// TIA Portal V17 export
// export: Created 2022-03-12T16:05:15.1481305Z, ExportSetting WithDefaults, DisplayName Totally Integrated Automation Portal, DisplayVersion V17, DisplayName TIA Portal Openness, DisplayVersion V17, DisplayName TIA Portal Version Control Interface, DisplayVersion V17, DisplayName STEP 7 Professional, DisplayVersion V17, DisplayName STEP 7 Safety, DisplayVersion V17, DisplayName WinCC Advanced / Unified PC, DisplayVersion V17
FUNCTION_BLOCK "UN_02_PackML"   // FB31622, LAD
TITLE = UN_02_PackML
{ S7_Optimized_Access := 'TRUE' }
AUTHOR : tech.team.motioncontrol@siemens.com
FAMILY : CPG
VERSION : 1.0
// Support: tech.team.motioncontrol@siemens.com
// Fax: +49 (0) 9131/98-1297
// stored: AutoNumber true, IsIECCheckEnabled false, IsRetainMemResEnabled false, MemoryReserve 100, SetENOAutomatically false, UDAEnableTagReadback false
   VAR
      statLanguageSelectedOld { ExternalAccessible := 'False'; ExternalVisible := 'False'; ExternalWritable := 'False'} : Int := -1;
      statPackML_CMD_SC { ExternalAccessible := 'False'; ExternalVisible := 'False'; ExternalWritable := 'False'} : Bool;
      instUnitModeStateManager { ExternalAccessible := 'False'; ExternalVisible := 'False'; ExternalWritable := 'False'; S7_SetPoint := 'True'} : "LPMLV30_UnitModeStateManager";
      instUnitModeStateTimes { ExternalAccessible := 'False'; ExternalVisible := 'False'; ExternalWritable := 'False'; S7_SetPoint := 'True'} : "LPMLV30_UnitModeStateTimes";
      statRemoteCommand_ModeChangeRequest { ExternalAccessible := 'False'; ExternalVisible := 'False'; ExternalWritable := 'False'} : Struct
         Production { ExternalAccessible := 'False'; ExternalVisible := 'False'; ExternalWritable := 'False'} : Bool;   // Request to goto mode - PRODUCTION (mode #1)
         Maintenance { ExternalAccessible := 'False'; ExternalVisible := 'False'; ExternalWritable := 'False'} : Bool;   // Request to goto mode - MAINTENANCE (mode #2)
         Manual { ExternalAccessible := 'False'; ExternalVisible := 'False'; ExternalWritable := 'False'} : Bool;   // Request to goto mode - MANUAL (mode #3)
         UserMode01 { ExternalAccessible := 'False'; ExternalVisible := 'False'; ExternalWritable := 'False'} : Bool;   // Request to goto mode - USER MODE 01 (mode #4)
         UserMode02 { ExternalAccessible := 'False'; ExternalVisible := 'False'; ExternalWritable := 'False'} : Bool;   // Request to goto mode - USER MODE 02 (mode #5)
         UserMode03 { ExternalAccessible := 'False'; ExternalVisible := 'False'; ExternalWritable := 'False'} : Bool;   // Request to goto mode - USER MODE 03 (mode #6)
         UserMode04 { ExternalAccessible := 'False'; ExternalVisible := 'False'; ExternalWritable := 'False'} : Bool;   // Request to goto mode - USER MODE 04 (mode #7)
         UserMode05 { ExternalAccessible := 'False'; ExternalVisible := 'False'; ExternalWritable := 'False'} : Bool;   // Request to goto mode - USER MODE 05 (mode #8)
         UserMode06 { ExternalAccessible := 'False'; ExternalVisible := 'False'; ExternalWritable := 'False'} : Bool;   // Request to goto mode - USER MODE 06 (mode #9)
         UserMode07 { ExternalAccessible := 'False'; ExternalVisible := 'False'; ExternalWritable := 'False'} : Bool;   // Request to goto mode - USER MODE 07 (mode #10)
         UserMode08 { ExternalAccessible := 'False'; ExternalVisible := 'False'; ExternalWritable := 'False'} : Bool;   // Request to goto mode - USER MODE 08 (mode #11)
      END_STRUCT;
      TPResettingDelay { ExternalAccessible := 'False'; ExternalVisible := 'False'; ExternalWritable := 'False'; S7_SetPoint := 'True'} : TP_TIME;
      TPClearingDelay { ExternalAccessible := 'False'; ExternalVisible := 'False'; ExternalWritable := 'False'; S7_SetPoint := 'True'} : TP_TIME;
   END_VAR
   VAR_TEMP
      tempDiagnosticsBufferIndexForHMI : Int;   // Temporary integer for PackML HMI diagnostics
   END_VAR
   VAR_TEMP   // added for the SCL form of the ladder/FBD networks
      _w1 : Bool;
   END_VAR
BEGIN

REGION Network 1: PackML ModeManager & State Model - Reset command
   // Reset Command:
   // If the machine is stopped and there are no faults (no stop or abort commands), 
   // then automatically reset and move the machine to idle.  This is common when all 
   // the faults are cleared in the Clearing state and the machine moves to the 
   // Stopped state with no more faults.
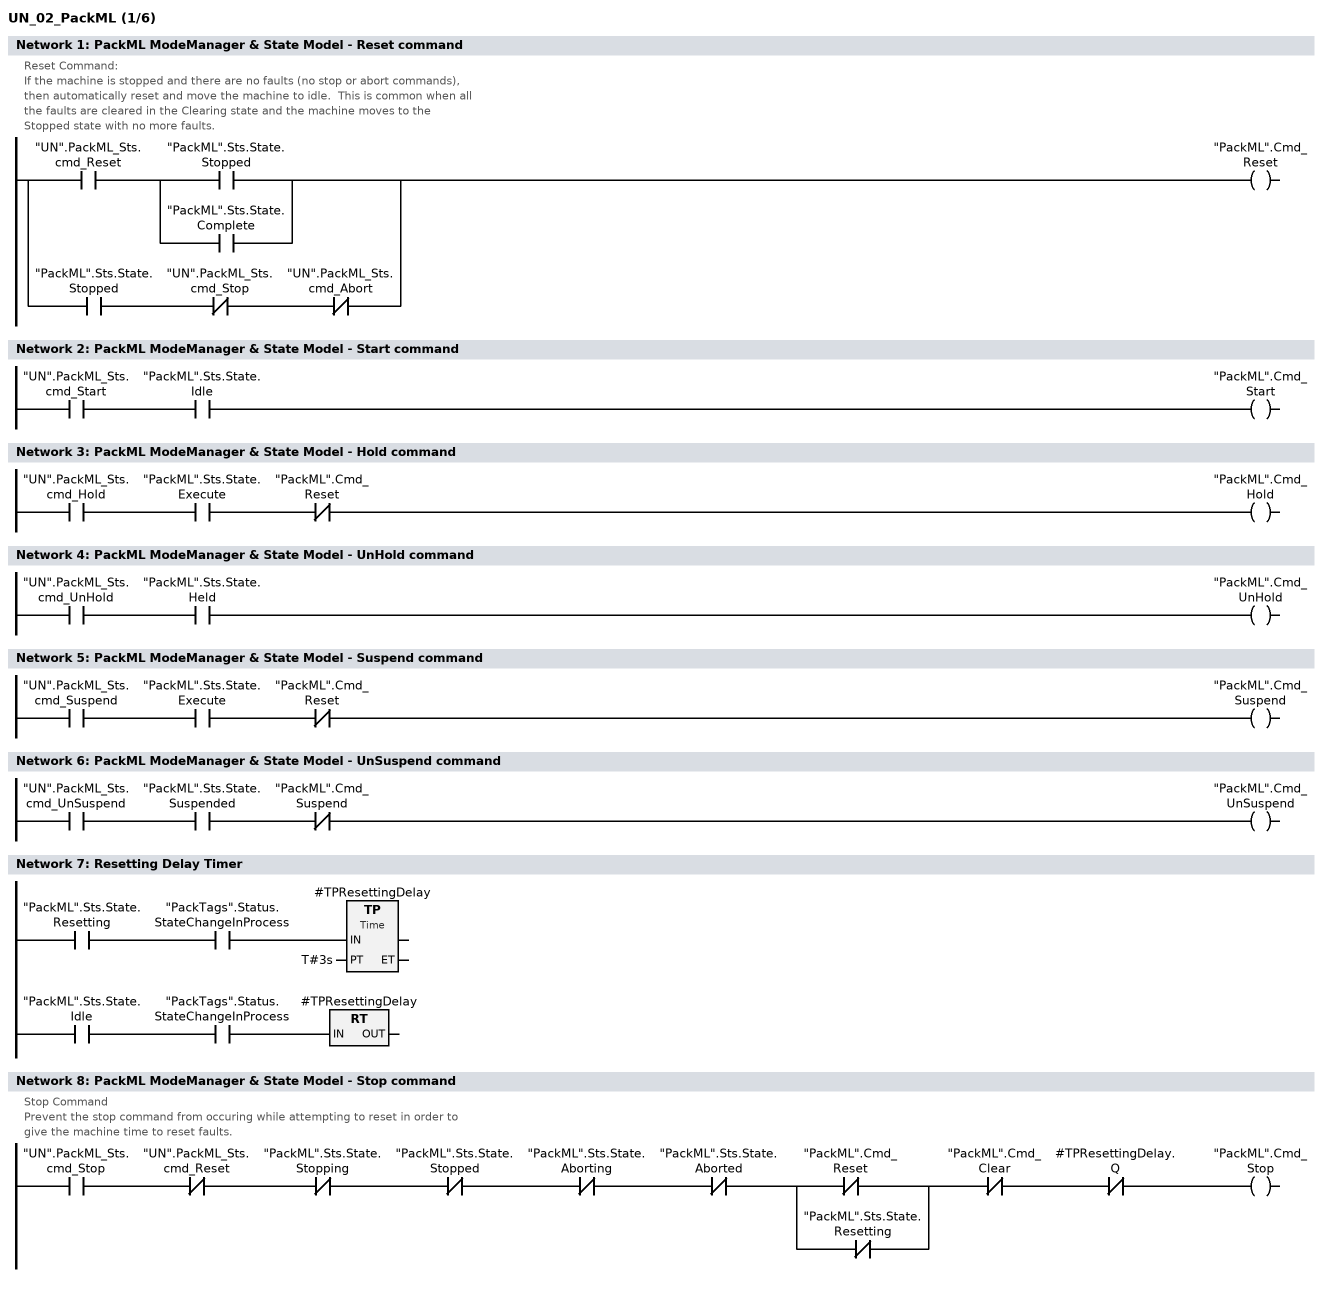
   RUNG wire#powerrail
      Contact( "UN".PackML_Sts.cmd_Reset )
      wire#w1
      Contact( "PackML".Sts.State.Stopped )
      wire#w2
      Coil( "PackML".Cmd_Reset )
   END_RUNG
   RUNG wire#w1
      Contact( "PackML".Sts.State.Complete )
   END_RUNG wire#w2
   RUNG wire#powerrail
      Contact( "PackML".Sts.State.Stopped )
      I_Contact( "UN".PackML_Sts.cmd_Stop )
      I_Contact( "UN".PackML_Sts.cmd_Abort )
   END_RUNG wire#w2
   // the same network as SCL:
   "PackML".Cmd_Reset := ("UN".PackML_Sts.cmd_Reset AND ("PackML".Sts.State.Stopped OR "PackML".Sts.State.Complete)) OR ("PackML".Sts.State.Stopped AND NOT "UN".PackML_Sts.cmd_Stop AND NOT "UN".PackML_Sts.cmd_Abort);
END_REGION

REGION Network 2: PackML ModeManager & State Model - Start command
   RUNG wire#powerrail
      Contact( "UN".PackML_Sts.cmd_Start )
      Contact( "PackML".Sts.State.Idle )
      Coil( "PackML".Cmd_Start )
   END_RUNG
   // the same network as SCL:
   "PackML".Cmd_Start := "UN".PackML_Sts.cmd_Start AND "PackML".Sts.State.Idle;
END_REGION

REGION Network 3: PackML ModeManager & State Model - Hold command
   RUNG wire#powerrail
      Contact( "UN".PackML_Sts.cmd_Hold )
      Contact( "PackML".Sts.State.Execute )
      I_Contact( "PackML".Cmd_Reset )
      Coil( "PackML".Cmd_Hold )
   END_RUNG
   // the same network as SCL:
   "PackML".Cmd_Hold := "UN".PackML_Sts.cmd_Hold AND "PackML".Sts.State.Execute AND NOT "PackML".Cmd_Reset;
END_REGION

REGION Network 4: PackML ModeManager & State Model - UnHold command
   RUNG wire#powerrail
      Contact( "UN".PackML_Sts.cmd_UnHold )
      Contact( "PackML".Sts.State.Held )
      Coil( "PackML".Cmd_UnHold )
   END_RUNG
   // the same network as SCL:
   "PackML".Cmd_UnHold := "UN".PackML_Sts.cmd_UnHold AND "PackML".Sts.State.Held;
END_REGION

REGION Network 5: PackML ModeManager & State Model - Suspend command
   RUNG wire#powerrail
      Contact( "UN".PackML_Sts.cmd_Suspend )
      Contact( "PackML".Sts.State.Execute )
      I_Contact( "PackML".Cmd_Reset )
      Coil( "PackML".Cmd_Suspend )
   END_RUNG
   // the same network as SCL:
   "PackML".Cmd_Suspend := "UN".PackML_Sts.cmd_Suspend AND "PackML".Sts.State.Execute AND NOT "PackML".Cmd_Reset;
END_REGION

REGION Network 6: PackML ModeManager & State Model - UnSuspend command
   RUNG wire#powerrail
      Contact( "UN".PackML_Sts.cmd_UnSuspend )
      Contact( "PackML".Sts.State.Suspended )
      I_Contact( "PackML".Cmd_Suspend )
      Coil( "PackML".Cmd_UnSuspend )
   END_RUNG
   // the same network as SCL:
   "PackML".Cmd_UnSuspend := "UN".PackML_Sts.cmd_UnSuspend AND "PackML".Sts.State.Suspended AND NOT "PackML".Cmd_Suspend;
END_REGION

REGION Network 7: Resetting Delay Timer
   RUNG wire#powerrail
      Contact( "PackML".Sts.State.Resetting )
      Contact( "PackTags".Status.StateChangeInProcess )
      { S7_Templates := "time_type := Time" } #TPResettingDelay.TP(pt := T#3s, et =>)
   END_RUNG
   RUNG wire#powerrail
      Contact( "PackML".Sts.State.Idle )
      Contact( "PackTags".Status.StateChangeInProcess )
      RT_Coil( #TPResettingDelay )
   END_RUNG
   // the same network as SCL:
   #TPResettingDelay(IN := "PackML".Sts.State.Resetting AND "PackTags".Status.StateChangeInProcess, PT := T#3s);   // TP
   IF "PackML".Sts.State.Idle AND "PackTags".Status.StateChangeInProcess THEN
       RESET_TIMER(#TPResettingDelay);
   END_IF;
END_REGION

REGION Network 8: PackML ModeManager & State Model - Stop command
   // Stop Command
   // Prevent the stop command from occuring while attempting to reset in order to 
   // give the machine time to reset faults.
   RUNG wire#powerrail
      Contact( "UN".PackML_Sts.cmd_Stop )
      I_Contact( "UN".PackML_Sts.cmd_Reset )
      I_Contact( "PackML".Sts.State.Stopping )
      I_Contact( "PackML".Sts.State.Stopped )
      I_Contact( "PackML".Sts.State.Aborting )
      I_Contact( "PackML".Sts.State.Aborted )
      wire#w1
      I_Contact( "PackML".Cmd_Reset )
      wire#w2
      I_Contact( "PackML".Cmd_Clear )
      I_Contact( #TPResettingDelay.Q )
      Coil( "PackML".Cmd_Stop )
   END_RUNG
   RUNG wire#w1
      I_Contact( "PackML".Sts.State.Resetting )
   END_RUNG wire#w2
   // the same network as SCL:
   "PackML".Cmd_Stop := "UN".PackML_Sts.cmd_Stop AND NOT "UN".PackML_Sts.cmd_Reset AND NOT "PackML".Sts.State.Stopping AND NOT "PackML".Sts.State.Stopped AND NOT "PackML".Sts.State.Aborting AND NOT "PackML".Sts.State.Aborted AND (NOT "PackML".Cmd_Reset OR NOT "PackML".Sts.State.Resetting) AND NOT "PackML".Cmd_Clear AND NOT #TPResettingDelay.Q;
END_REGION

REGION Network 9: Clearing Delay Timer
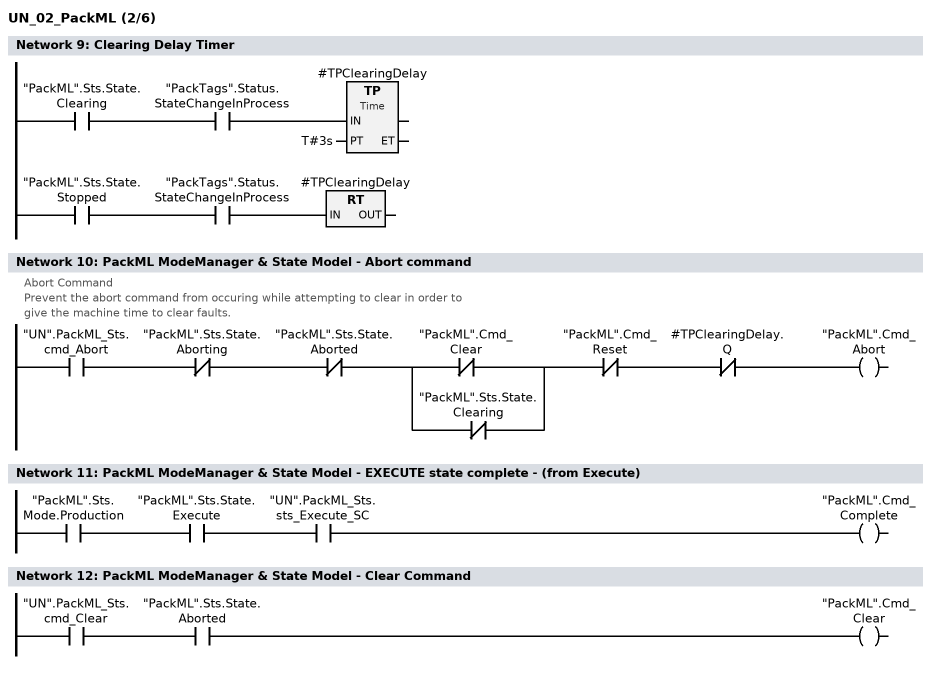
   RUNG wire#powerrail
      Contact( "PackML".Sts.State.Clearing )
      Contact( "PackTags".Status.StateChangeInProcess )
      { S7_Templates := "time_type := Time" } #TPClearingDelay.TP(pt := T#3s, et =>)
   END_RUNG
   RUNG wire#powerrail
      Contact( "PackML".Sts.State.Stopped )
      Contact( "PackTags".Status.StateChangeInProcess )
      RT_Coil( #TPClearingDelay )
   END_RUNG
   // the same network as SCL:
   #TPClearingDelay(IN := "PackML".Sts.State.Clearing AND "PackTags".Status.StateChangeInProcess, PT := T#3s);   // TP
   IF "PackML".Sts.State.Stopped AND "PackTags".Status.StateChangeInProcess THEN
       RESET_TIMER(#TPClearingDelay);
   END_IF;
END_REGION

REGION Network 10: PackML ModeManager & State Model - Abort command
   // Abort Command
   // Prevent the abort command from occuring while attempting to clear in order to 
   // give the machine time to clear faults.
   RUNG wire#powerrail
      Contact( "UN".PackML_Sts.cmd_Abort )
      I_Contact( "PackML".Sts.State.Aborting )
      I_Contact( "PackML".Sts.State.Aborted )
      wire#w1
      I_Contact( "PackML".Cmd_Clear )
      wire#w2
      I_Contact( "PackML".Cmd_Reset )
      I_Contact( #TPClearingDelay.Q )
      Coil( "PackML".Cmd_Abort )
   END_RUNG
   RUNG wire#w1
      I_Contact( "PackML".Sts.State.Clearing )
   END_RUNG wire#w2
   // the same network as SCL:
   "PackML".Cmd_Abort := "UN".PackML_Sts.cmd_Abort AND NOT "PackML".Sts.State.Aborting AND NOT "PackML".Sts.State.Aborted AND (NOT "PackML".Cmd_Clear OR NOT "PackML".Sts.State.Clearing) AND NOT "PackML".Cmd_Reset AND NOT #TPClearingDelay.Q;
END_REGION

REGION Network 11: PackML ModeManager & State Model - EXECUTE state complete - (from Execute)
   RUNG wire#powerrail
      Contact( "PackML".Sts.Mode.Production )
      Contact( "PackML".Sts.State.Execute )
      Contact( "UN".PackML_Sts.sts_Execute_SC )
      Coil( "PackML".Cmd_Complete )
   END_RUNG
   // the same network as SCL:
   "PackML".Cmd_Complete := "PackML".Sts.Mode.Production AND "PackML".Sts.State.Execute AND "UN".PackML_Sts.sts_Execute_SC;
END_REGION

REGION Network 12: PackML ModeManager & State Model - Clear Command
   RUNG wire#powerrail
      Contact( "UN".PackML_Sts.cmd_Clear )
      Contact( "PackML".Sts.State.Aborted )
      Coil( "PackML".Cmd_Clear )
   END_RUNG
   // the same network as SCL:
   "PackML".Cmd_Clear := "UN".PackML_Sts.cmd_Clear AND "PackML".Sts.State.Aborted;
END_REGION

REGION Network 13: External PackML Mode Commands
   // External State Commands are handled in the UN_05_EventControl routine to ensure that the unit machine level alarm manager captures the reason for any machine stoppage.
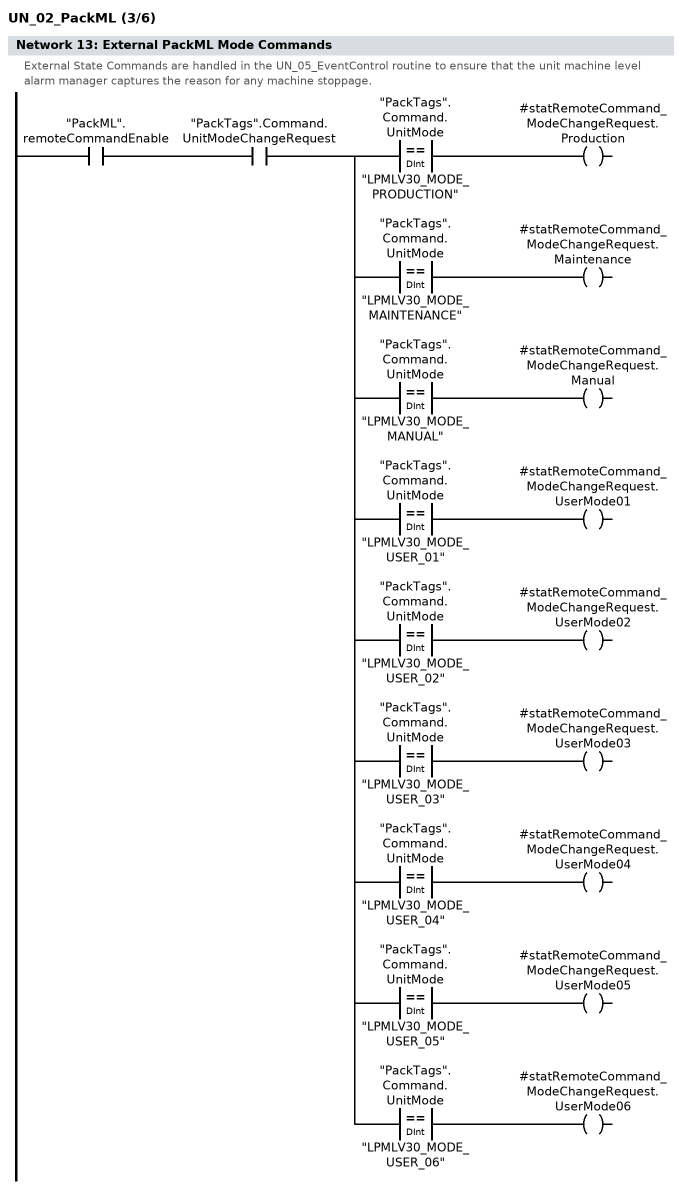
   RUNG wire#powerrail
      Contact( "PackML".remoteCommandEnable )
      Contact( "PackTags".Command.UnitModeChangeRequest )
      wire#w1
      { S7_Templates := "SrcType := DInt" } EQ_Contact(in1 := "PackTags".Command.UnitMode, in2 := "LPMLV30_MODE_PRODUCTION")
      Coil( #statRemoteCommand_ModeChangeRequest.Production )
   END_RUNG
   RUNG wire#w1
      { S7_Templates := "SrcType := DInt" } EQ_Contact(in1 := "PackTags".Command.UnitMode, in2 := "LPMLV30_MODE_MAINTENANCE")
      Coil( #statRemoteCommand_ModeChangeRequest.Maintenance )
   END_RUNG
   RUNG wire#w1
      { S7_Templates := "SrcType := DInt" } EQ_Contact(in1 := "PackTags".Command.UnitMode, in2 := "LPMLV30_MODE_MANUAL")
      Coil( #statRemoteCommand_ModeChangeRequest.Manual )
   END_RUNG
   RUNG wire#w1
      { S7_Templates := "SrcType := DInt" } EQ_Contact(in1 := "PackTags".Command.UnitMode, in2 := "LPMLV30_MODE_USER_01")
      Coil( #statRemoteCommand_ModeChangeRequest.UserMode01 )
   END_RUNG
   RUNG wire#w1
      { S7_Templates := "SrcType := DInt" } EQ_Contact(in1 := "PackTags".Command.UnitMode, in2 := "LPMLV30_MODE_USER_02")
      Coil( #statRemoteCommand_ModeChangeRequest.UserMode02 )
   END_RUNG
   RUNG wire#w1
      { S7_Templates := "SrcType := DInt" } EQ_Contact(in1 := "PackTags".Command.UnitMode, in2 := "LPMLV30_MODE_USER_03")
      Coil( #statRemoteCommand_ModeChangeRequest.UserMode03 )
   END_RUNG
   RUNG wire#w1
      { S7_Templates := "SrcType := DInt" } EQ_Contact(in1 := "PackTags".Command.UnitMode, in2 := "LPMLV30_MODE_USER_04")
      Coil( #statRemoteCommand_ModeChangeRequest.UserMode04 )
   END_RUNG
   RUNG wire#w1
      { S7_Templates := "SrcType := DInt" } EQ_Contact(in1 := "PackTags".Command.UnitMode, in2 := "LPMLV30_MODE_USER_05")
      Coil( #statRemoteCommand_ModeChangeRequest.UserMode05 )
   END_RUNG
   RUNG wire#w1
      { S7_Templates := "SrcType := DInt" } EQ_Contact(in1 := "PackTags".Command.UnitMode, in2 := "LPMLV30_MODE_USER_06")
      Coil( #statRemoteCommand_ModeChangeRequest.UserMode06 )
   END_RUNG
   // the same network as SCL:
   #_w1 := "PackML".remoteCommandEnable AND "PackTags".Command.UnitModeChangeRequest;
   #statRemoteCommand_ModeChangeRequest.Production := #_w1 AND ("PackTags".Command.UnitMode = "LPMLV30_MODE_PRODUCTION");
   #statRemoteCommand_ModeChangeRequest.Maintenance := #_w1 AND ("PackTags".Command.UnitMode = "LPMLV30_MODE_MAINTENANCE");
   #statRemoteCommand_ModeChangeRequest.Manual := #_w1 AND ("PackTags".Command.UnitMode = "LPMLV30_MODE_MANUAL");
   #statRemoteCommand_ModeChangeRequest.UserMode01 := #_w1 AND ("PackTags".Command.UnitMode = "LPMLV30_MODE_USER_01");
   #statRemoteCommand_ModeChangeRequest.UserMode02 := #_w1 AND ("PackTags".Command.UnitMode = "LPMLV30_MODE_USER_02");
   #statRemoteCommand_ModeChangeRequest.UserMode03 := #_w1 AND ("PackTags".Command.UnitMode = "LPMLV30_MODE_USER_03");
   #statRemoteCommand_ModeChangeRequest.UserMode04 := #_w1 AND ("PackTags".Command.UnitMode = "LPMLV30_MODE_USER_04");
   #statRemoteCommand_ModeChangeRequest.UserMode05 := #_w1 AND ("PackTags".Command.UnitMode = "LPMLV30_MODE_USER_05");
   #statRemoteCommand_ModeChangeRequest.UserMode06 := #_w1 AND ("PackTags".Command.UnitMode = "LPMLV30_MODE_USER_06");
END_REGION

REGION Network 14: Call thePackML Mode Manager & State Model FB
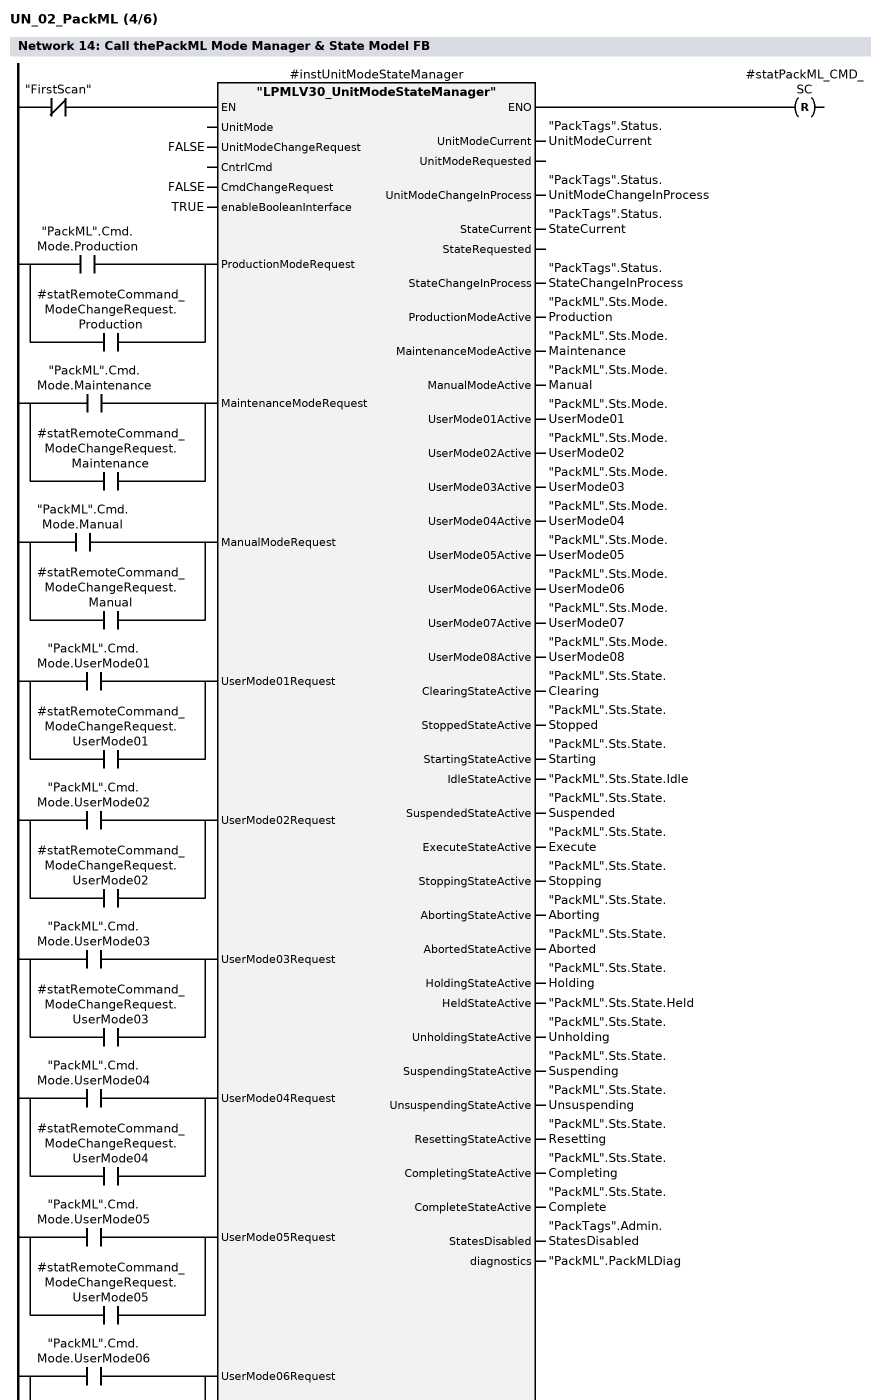
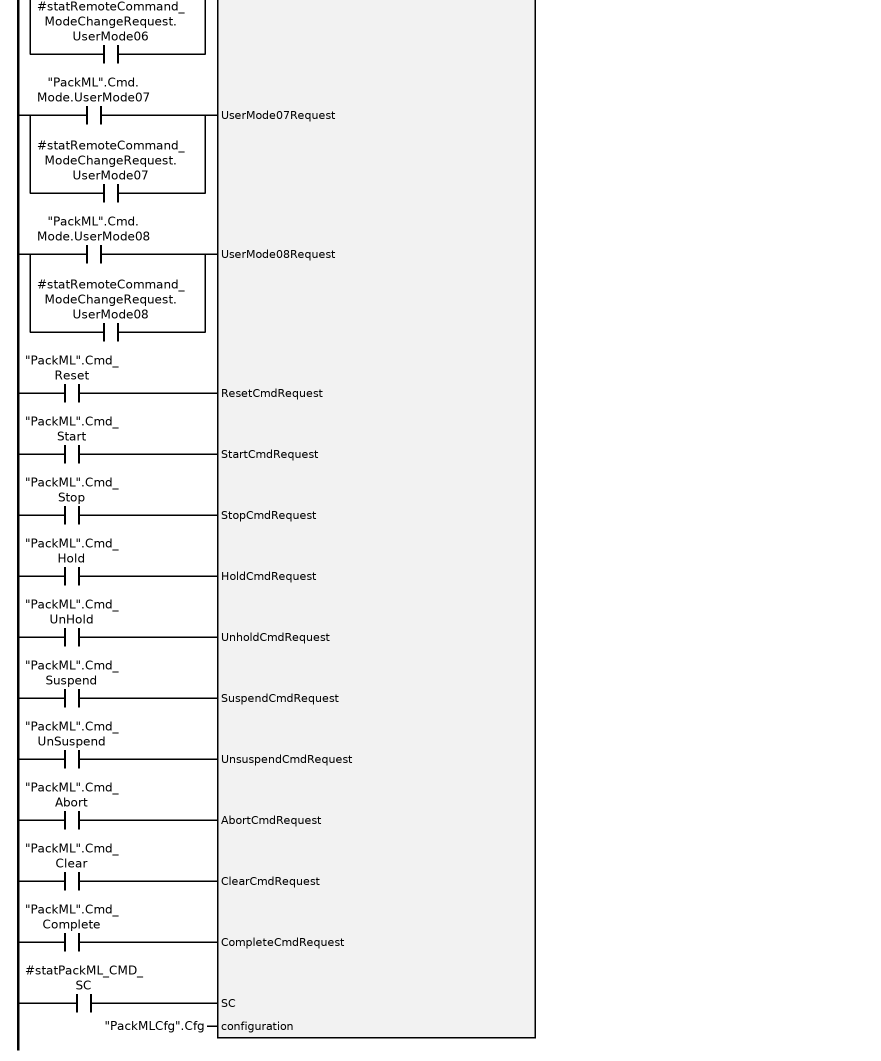
   RUNG wire#powerrail
      I_Contact( "FirstScan" )
      #instUnitModeStateManager(ProductionModeRequest := wire#w1, MaintenanceModeRequest := wire#w2, ManualModeRequest := wire#w3, UserMode01Request := wire#w4, UserMode02Request := wire#w5, UserMode03Request := wire#w6, UserMode04Request := wire#w7, UserMode05Request := wire#w8, UserMode06Request := wire#w9, UserMode07Request := wire#w10, UserMode08Request := wire#w11, ResetCmdRequest := wire#w12, StartCmdRequest := wire#w13, StopCmdRequest := wire#w14, HoldCmdRequest := wire#w15, UnholdCmdRequest := wire#w16, SuspendCmdRequest := wire#w17, UnsuspendCmdRequest := wire#w18, AbortCmdRequest := wire#w19, ClearCmdRequest := wire#w20, CompleteCmdRequest := wire#w21, SC := wire#w22, UnitMode :=, UnitModeChangeRequest := FALSE, CntrlCmd :=, CmdChangeRequest := FALSE, enableBooleanInterface := TRUE, configuration := "PackMLCfg".Cfg, UnitModeCurrent => "PackTags".Status.UnitModeCurrent, UnitModeRequested =>, UnitModeChangeInProcess => "PackTags".Status.UnitModeChangeInProcess, StateCurrent => "PackTags".Status.StateCurrent, StateRequested =>, StateChangeInProcess => "PackTags".Status.StateChangeInProcess, ProductionModeActive => "PackML".Sts.Mode.Production, MaintenanceModeActive => "PackML".Sts.Mode.Maintenance, ManualModeActive => "PackML".Sts.Mode.Manual, UserMode01Active => "PackML".Sts.Mode.UserMode01, UserMode02Active => "PackML".Sts.Mode.UserMode02, UserMode03Active => "PackML".Sts.Mode.UserMode03, UserMode04Active => "PackML".Sts.Mode.UserMode04, UserMode05Active => "PackML".Sts.Mode.UserMode05, UserMode06Active => "PackML".Sts.Mode.UserMode06, UserMode07Active => "PackML".Sts.Mode.UserMode07, UserMode08Active => "PackML".Sts.Mode.UserMode08, ClearingStateActive => "PackML".Sts.State.Clearing, StoppedStateActive => "PackML".Sts.State.Stopped, StartingStateActive => "PackML".Sts.State.Starting, IdleStateActive => "PackML".Sts.State.Idle, SuspendedStateActive => "PackML".Sts.State.Suspended, ExecuteStateActive => "PackML".Sts.State.Execute, StoppingStateActive => "PackML".Sts.State.Stopping, AbortingStateActive => "PackML".Sts.State.Aborting, AbortedStateActive => "PackML".Sts.State.Aborted, HoldingStateActive => "PackML".Sts.State.Holding, HeldStateActive => "PackML".Sts.State.Held, UnholdingStateActive => "PackML".Sts.State.Unholding, SuspendingStateActive => "PackML".Sts.State.Suspending, UnsuspendingStateActive => "PackML".Sts.State.Unsuspending, ResettingStateActive => "PackML".Sts.State.Resetting, CompletingStateActive => "PackML".Sts.State.Completing, CompleteStateActive => "PackML".Sts.State.Complete, StatesDisabled => "PackTags".Admin.StatesDisabled, diagnostics => "PackML".PackMLDiag)
      R_Coil( #statPackML_CMD_SC )
   END_RUNG
   RUNG wire#powerrail
      Contact( "PackML".Cmd.Mode.Production )
   END_RUNG wire#w1
   RUNG wire#powerrail
      Contact( #statRemoteCommand_ModeChangeRequest.Production )
   END_RUNG wire#w1
   RUNG wire#powerrail
      Contact( "PackML".Cmd.Mode.Maintenance )
   END_RUNG wire#w2
   RUNG wire#powerrail
      Contact( #statRemoteCommand_ModeChangeRequest.Maintenance )
   END_RUNG wire#w2
   RUNG wire#powerrail
      Contact( "PackML".Cmd.Mode.Manual )
   END_RUNG wire#w3
   RUNG wire#powerrail
      Contact( #statRemoteCommand_ModeChangeRequest.Manual )
   END_RUNG wire#w3
   RUNG wire#powerrail
      Contact( "PackML".Cmd.Mode.UserMode01 )
   END_RUNG wire#w4
   RUNG wire#powerrail
      Contact( #statRemoteCommand_ModeChangeRequest.UserMode01 )
   END_RUNG wire#w4
   RUNG wire#powerrail
      Contact( "PackML".Cmd.Mode.UserMode02 )
   END_RUNG wire#w5
   RUNG wire#powerrail
      Contact( #statRemoteCommand_ModeChangeRequest.UserMode02 )
   END_RUNG wire#w5
   RUNG wire#powerrail
      Contact( "PackML".Cmd.Mode.UserMode03 )
   END_RUNG wire#w6
   RUNG wire#powerrail
      Contact( #statRemoteCommand_ModeChangeRequest.UserMode03 )
   END_RUNG wire#w6
   RUNG wire#powerrail
      Contact( "PackML".Cmd.Mode.UserMode04 )
   END_RUNG wire#w7
   RUNG wire#powerrail
      Contact( #statRemoteCommand_ModeChangeRequest.UserMode04 )
   END_RUNG wire#w7
   RUNG wire#powerrail
      Contact( "PackML".Cmd.Mode.UserMode05 )
   END_RUNG wire#w8
   RUNG wire#powerrail
      Contact( #statRemoteCommand_ModeChangeRequest.UserMode05 )
   END_RUNG wire#w8
   RUNG wire#powerrail
      Contact( "PackML".Cmd.Mode.UserMode06 )
   END_RUNG wire#w9
   RUNG wire#powerrail
      Contact( #statRemoteCommand_ModeChangeRequest.UserMode06 )
   END_RUNG wire#w9
   RUNG wire#powerrail
      Contact( "PackML".Cmd.Mode.UserMode07 )
   END_RUNG wire#w10
   RUNG wire#powerrail
      Contact( #statRemoteCommand_ModeChangeRequest.UserMode07 )
   END_RUNG wire#w10
   RUNG wire#powerrail
      Contact( "PackML".Cmd.Mode.UserMode08 )
   END_RUNG wire#w11
   RUNG wire#powerrail
      Contact( #statRemoteCommand_ModeChangeRequest.UserMode08 )
   END_RUNG wire#w11
   RUNG wire#powerrail
      Contact( "PackML".Cmd_Reset )
   END_RUNG wire#w12
   RUNG wire#powerrail
      Contact( "PackML".Cmd_Start )
   END_RUNG wire#w13
   RUNG wire#powerrail
      Contact( "PackML".Cmd_Stop )
   END_RUNG wire#w14
   RUNG wire#powerrail
      Contact( "PackML".Cmd_Hold )
   END_RUNG wire#w15
   RUNG wire#powerrail
      Contact( "PackML".Cmd_UnHold )
   END_RUNG wire#w16
   RUNG wire#powerrail
      Contact( "PackML".Cmd_Suspend )
   END_RUNG wire#w17
   RUNG wire#powerrail
      Contact( "PackML".Cmd_UnSuspend )
   END_RUNG wire#w18
   RUNG wire#powerrail
      Contact( "PackML".Cmd_Abort )
   END_RUNG wire#w19
   RUNG wire#powerrail
      Contact( "PackML".Cmd_Clear )
   END_RUNG wire#w20
   RUNG wire#powerrail
      Contact( "PackML".Cmd_Complete )
   END_RUNG wire#w21
   RUNG wire#powerrail
      Contact( #statPackML_CMD_SC )
   END_RUNG wire#w22
   // the same network as SCL:
   #instUnitModeStateManager(EN := NOT "FirstScan",   // "LPMLV30_UnitModeStateManager"
                           UnitModeChangeRequest := FALSE,
                           CmdChangeRequest := FALSE,
                           enableBooleanInterface := TRUE,
                           ProductionModeRequest := "PackML".Cmd.Mode.Production OR #statRemoteCommand_ModeChangeRequest.Production,
                           MaintenanceModeRequest := "PackML".Cmd.Mode.Maintenance OR #statRemoteCommand_ModeChangeRequest.Maintenance,
                           ManualModeRequest := "PackML".Cmd.Mode.Manual OR #statRemoteCommand_ModeChangeRequest.Manual,
                           UserMode01Request := "PackML".Cmd.Mode.UserMode01 OR #statRemoteCommand_ModeChangeRequest.UserMode01,
                           UserMode02Request := "PackML".Cmd.Mode.UserMode02 OR #statRemoteCommand_ModeChangeRequest.UserMode02,
                           UserMode03Request := "PackML".Cmd.Mode.UserMode03 OR #statRemoteCommand_ModeChangeRequest.UserMode03,
                           UserMode04Request := "PackML".Cmd.Mode.UserMode04 OR #statRemoteCommand_ModeChangeRequest.UserMode04,
                           UserMode05Request := "PackML".Cmd.Mode.UserMode05 OR #statRemoteCommand_ModeChangeRequest.UserMode05,
                           UserMode06Request := "PackML".Cmd.Mode.UserMode06 OR #statRemoteCommand_ModeChangeRequest.UserMode06,
                           UserMode07Request := "PackML".Cmd.Mode.UserMode07 OR #statRemoteCommand_ModeChangeRequest.UserMode07,
                           UserMode08Request := "PackML".Cmd.Mode.UserMode08 OR #statRemoteCommand_ModeChangeRequest.UserMode08,
                           ResetCmdRequest := "PackML".Cmd_Reset,
                           StartCmdRequest := "PackML".Cmd_Start,
                           StopCmdRequest := "PackML".Cmd_Stop,
                           HoldCmdRequest := "PackML".Cmd_Hold,
                           UnholdCmdRequest := "PackML".Cmd_UnHold,
                           SuspendCmdRequest := "PackML".Cmd_Suspend,
                           UnsuspendCmdRequest := "PackML".Cmd_UnSuspend,
                           AbortCmdRequest := "PackML".Cmd_Abort,
                           ClearCmdRequest := "PackML".Cmd_Clear,
                           CompleteCmdRequest := "PackML".Cmd_Complete,
                           SC := #statPackML_CMD_SC,
                           configuration := "PackMLCfg".Cfg,
                           UnitModeCurrent => "PackTags".Status.UnitModeCurrent,
                           UnitModeChangeInProcess => "PackTags".Status.UnitModeChangeInProcess,
                           StateCurrent => "PackTags".Status.StateCurrent,
                           StateChangeInProcess => "PackTags".Status.StateChangeInProcess,
                           ProductionModeActive => "PackML".Sts.Mode.Production,
                           MaintenanceModeActive => "PackML".Sts.Mode.Maintenance,
                           ManualModeActive => "PackML".Sts.Mode.Manual,
                           UserMode01Active => "PackML".Sts.Mode.UserMode01,
                           UserMode02Active => "PackML".Sts.Mode.UserMode02,
                           UserMode03Active => "PackML".Sts.Mode.UserMode03,
                           UserMode04Active => "PackML".Sts.Mode.UserMode04,
                           UserMode05Active => "PackML".Sts.Mode.UserMode05,
                           UserMode06Active => "PackML".Sts.Mode.UserMode06,
                           UserMode07Active => "PackML".Sts.Mode.UserMode07,
                           UserMode08Active => "PackML".Sts.Mode.UserMode08,
                           ClearingStateActive => "PackML".Sts.State.Clearing,
                           StoppedStateActive => "PackML".Sts.State.Stopped,
                           StartingStateActive => "PackML".Sts.State.Starting,
                           IdleStateActive => "PackML".Sts.State.Idle,
                           SuspendedStateActive => "PackML".Sts.State.Suspended,
                           ExecuteStateActive => "PackML".Sts.State.Execute,
                           StoppingStateActive => "PackML".Sts.State.Stopping,
                           AbortingStateActive => "PackML".Sts.State.Aborting,
                           AbortedStateActive => "PackML".Sts.State.Aborted,
                           HoldingStateActive => "PackML".Sts.State.Holding,
                           HeldStateActive => "PackML".Sts.State.Held,
                           UnholdingStateActive => "PackML".Sts.State.Unholding,
                           SuspendingStateActive => "PackML".Sts.State.Suspending,
                           UnsuspendingStateActive => "PackML".Sts.State.Unsuspending,
                           ResettingStateActive => "PackML".Sts.State.Resetting,
                           CompletingStateActive => "PackML".Sts.State.Completing,
                           CompleteStateActive => "PackML".Sts.State.Complete,
                           StatesDisabled => "PackTags".Admin.StatesDisabled,
                           diagnostics => "PackML".PackMLDiag,
                           ENO => #_w1);
   IF #_w1 THEN #statPackML_CMD_SC := FALSE; END_IF;
END_REGION

REGION Network 15: "Times" used to format PackML.Admin times and for the HMI display
   // PackML State and Mode Times for HMI
   // 
   // The times spent in each mode and state are calculated in the PackML FB.  This 
   // FB is used to move the modes and states time arrays (current and cumulative 
   // times) into a single array - that is based upon the curent mode - for both 
   // current and cumlative state times.   This single arry is used by the HMI
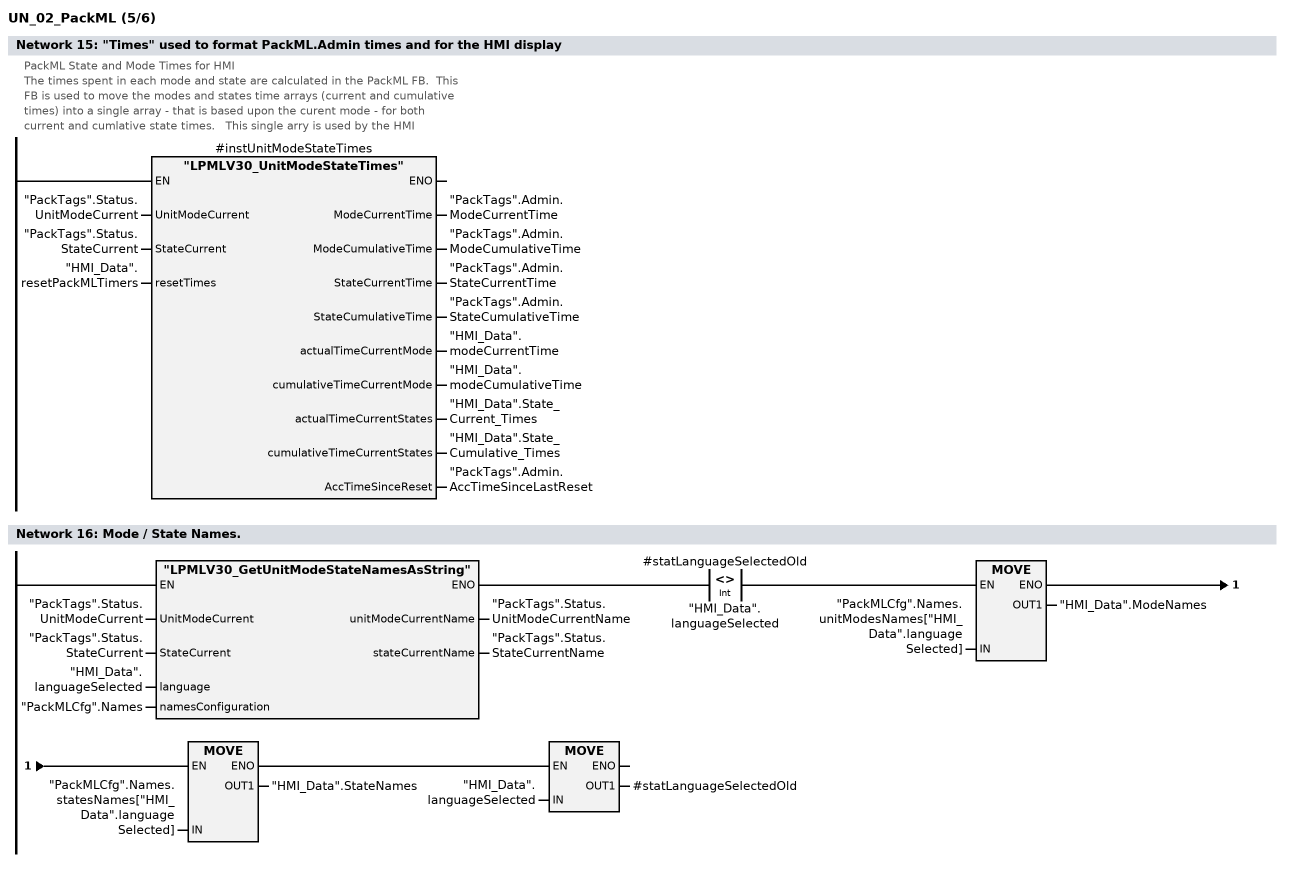
   RUNG wire#powerrail
      #instUnitModeStateTimes(UnitModeCurrent := "PackTags".Status.UnitModeCurrent, StateCurrent := "PackTags".Status.StateCurrent, resetTimes := "HMI_Data".resetPackMLTimers, ModeCurrentTime => "PackTags".Admin.ModeCurrentTime, ModeCumulativeTime => "PackTags".Admin.ModeCumulativeTime, StateCurrentTime => "PackTags".Admin.StateCurrentTime, StateCumulativeTime => "PackTags".Admin.StateCumulativeTime, actualTimeCurrentMode => "HMI_Data".modeCurrentTime, cumulativeTimeCurrentMode => "HMI_Data".modeCumulativeTime, actualTimeCurrentStates => "HMI_Data".State_Current_Times, cumulativeTimeCurrentStates => "HMI_Data".State_Cumulative_Times, AccTimeSinceReset => "PackTags".Admin.AccTimeSinceLastReset)
   END_RUNG
   // the same network as SCL:
   #instUnitModeStateTimes(UnitModeCurrent := "PackTags".Status.UnitModeCurrent,   // "LPMLV30_UnitModeStateTimes"
                           StateCurrent := "PackTags".Status.StateCurrent,
                           resetTimes := "HMI_Data".resetPackMLTimers,
                           ModeCurrentTime => "PackTags".Admin.ModeCurrentTime,
                           ModeCumulativeTime => "PackTags".Admin.ModeCumulativeTime,
                           StateCurrentTime => "PackTags".Admin.StateCurrentTime,
                           StateCumulativeTime => "PackTags".Admin.StateCumulativeTime,
                           actualTimeCurrentMode => "HMI_Data".modeCurrentTime,
                           cumulativeTimeCurrentMode => "HMI_Data".modeCumulativeTime,
                           actualTimeCurrentStates => "HMI_Data".State_Current_Times,
                           cumulativeTimeCurrentStates => "HMI_Data".State_Cumulative_Times,
                           AccTimeSinceReset => "PackTags".Admin.AccTimeSinceLastReset);
END_REGION

REGION Network 16: Mode / State Names.
   RUNG wire#powerrail
      "LPMLV30_GetUnitModeStateNamesAsString"(UnitModeCurrent := "PackTags".Status.UnitModeCurrent, StateCurrent := "PackTags".Status.StateCurrent, language := "HMI_Data".languageSelected, namesConfiguration := "PackMLCfg".Names, unitModeCurrentName => "PackTags".Status.UnitModeCurrentName, stateCurrentName => "PackTags".Status.StateCurrentName)
      { S7_Templates := "SrcType := Int" } NE_Contact(in1 := #statLanguageSelectedOld, in2 := "HMI_Data".languageSelected)
      Move(in := "PackMLCfg".Names.unitModesNames["HMI_Data".languageSelected], out1 => "HMI_Data".ModeNames)
      Move(in := "PackMLCfg".Names.statesNames["HMI_Data".languageSelected], out1 => "HMI_Data".StateNames)
      Move(in := "HMI_Data".languageSelected, out1 => #statLanguageSelectedOld)
   END_RUNG
   // the same network as SCL:
   "LPMLV30_GetUnitModeStateNamesAsString"(UnitModeCurrent := "PackTags".Status.UnitModeCurrent,
                           StateCurrent := "PackTags".Status.StateCurrent,
                           language := "HMI_Data".languageSelected,
                           namesConfiguration := "PackMLCfg".Names,
                           unitModeCurrentName => "PackTags".Status.UnitModeCurrentName,
                           stateCurrentName => "PackTags".Status.StateCurrentName,
                           ENO => #_w1);
   IF #_w1 AND (#statLanguageSelectedOld <> "HMI_Data".languageSelected) THEN
       "HMI_Data".ModeNames := "PackMLCfg".Names.unitModesNames["HMI_Data".languageSelected];
       "HMI_Data".StateNames := "PackMLCfg".Names.statesNames["HMI_Data".languageSelected];
       #statLanguageSelectedOld := "HMI_Data".languageSelected;
   END_IF;
END_REGION

REGION Network 17: State Complete Commands
END_REGION

REGION Network 18: Set the State Complete (SC) bit
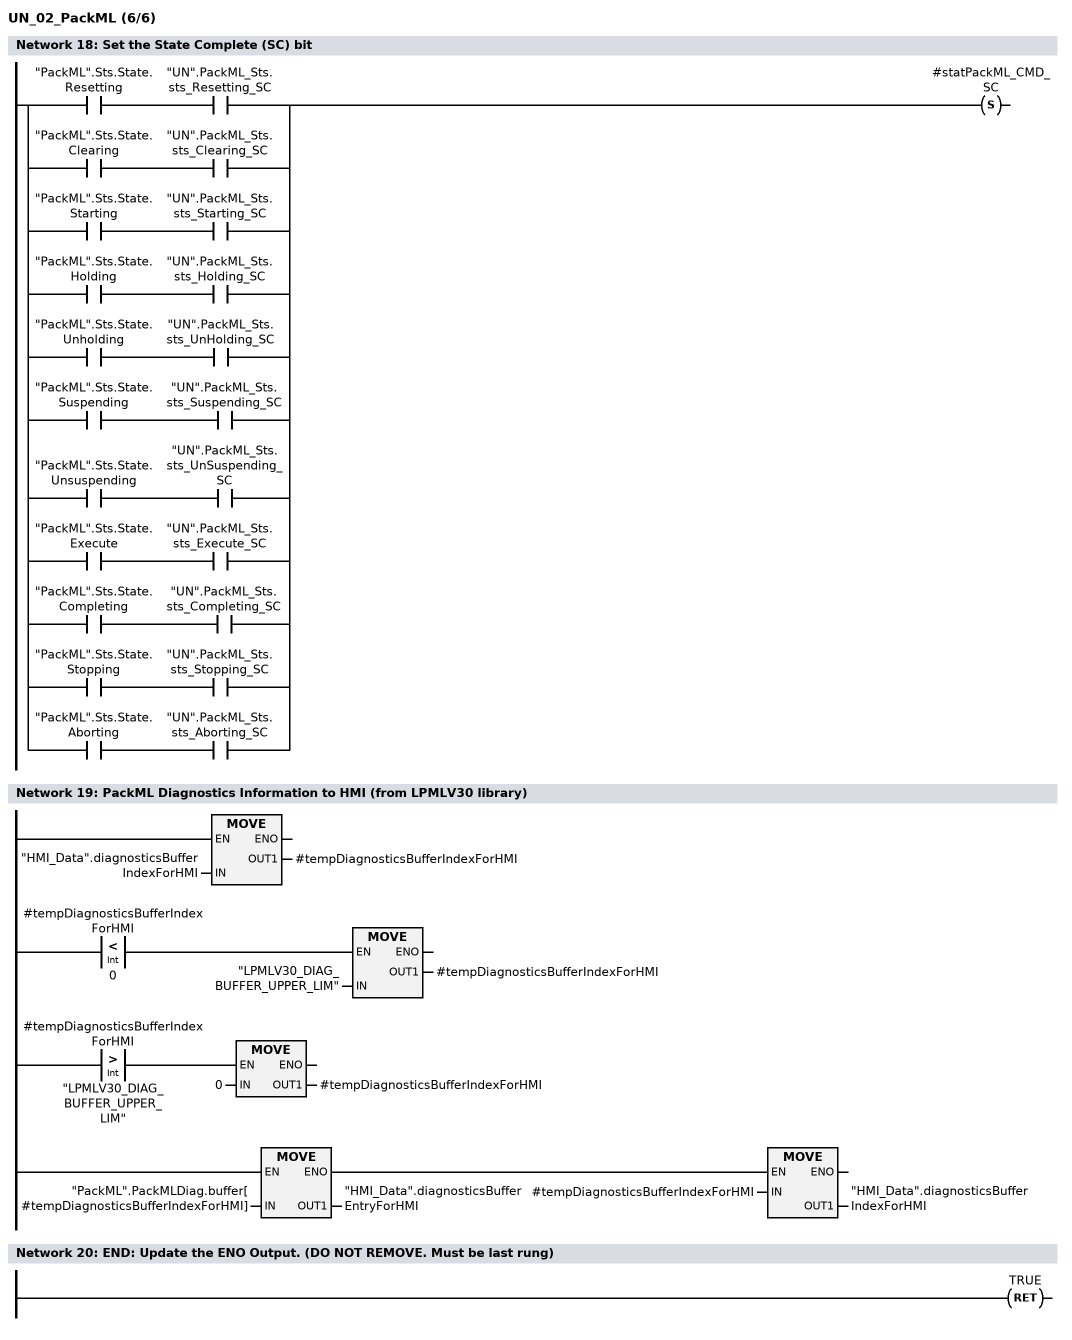
   RUNG wire#powerrail
      Contact( "PackML".Sts.State.Resetting )
      Contact( "UN".PackML_Sts.sts_Resetting_SC )
      wire#w1
      S_Coil( #statPackML_CMD_SC )
   END_RUNG
   RUNG wire#powerrail
      Contact( "PackML".Sts.State.Clearing )
      Contact( "UN".PackML_Sts.sts_Clearing_SC )
   END_RUNG wire#w1
   RUNG wire#powerrail
      Contact( "PackML".Sts.State.Starting )
      Contact( "UN".PackML_Sts.sts_Starting_SC )
   END_RUNG wire#w1
   RUNG wire#powerrail
      Contact( "PackML".Sts.State.Holding )
      Contact( "UN".PackML_Sts.sts_Holding_SC )
   END_RUNG wire#w1
   RUNG wire#powerrail
      Contact( "PackML".Sts.State.Unholding )
      Contact( "UN".PackML_Sts.sts_UnHolding_SC )
   END_RUNG wire#w1
   RUNG wire#powerrail
      Contact( "PackML".Sts.State.Suspending )
      Contact( "UN".PackML_Sts.sts_Suspending_SC )
   END_RUNG wire#w1
   RUNG wire#powerrail
      Contact( "PackML".Sts.State.Unsuspending )
      Contact( "UN".PackML_Sts.sts_UnSuspending_SC )
   END_RUNG wire#w1
   RUNG wire#powerrail
      Contact( "PackML".Sts.State.Execute )
      Contact( "UN".PackML_Sts.sts_Execute_SC )
   END_RUNG wire#w1
   RUNG wire#powerrail
      Contact( "PackML".Sts.State.Completing )
      Contact( "UN".PackML_Sts.sts_Completing_SC )
   END_RUNG wire#w1
   RUNG wire#powerrail
      Contact( "PackML".Sts.State.Stopping )
      Contact( "UN".PackML_Sts.sts_Stopping_SC )
   END_RUNG wire#w1
   RUNG wire#powerrail
      Contact( "PackML".Sts.State.Aborting )
      Contact( "UN".PackML_Sts.sts_Aborting_SC )
   END_RUNG wire#w1
   // the same network as SCL:
   IF ("PackML".Sts.State.Resetting AND "UN".PackML_Sts.sts_Resetting_SC) OR ("PackML".Sts.State.Clearing AND "UN".PackML_Sts.sts_Clearing_SC) OR ("PackML".Sts.State.Starting AND "UN".PackML_Sts.sts_Starting_SC) OR ("PackML".Sts.State.Holding AND "UN".PackML_Sts.sts_Holding_SC) OR ("PackML".Sts.State.Unholding AND "UN".PackML_Sts.sts_UnHolding_SC) OR ("PackML".Sts.State.Suspending AND "UN".PackML_Sts.sts_Suspending_SC) OR ("PackML".Sts.State.Unsuspending AND "UN".PackML_Sts.sts_UnSuspending_SC) OR ("PackML".Sts.State.Execute AND "UN".PackML_Sts.sts_Execute_SC) OR ("PackML".Sts.State.Completing AND "UN".PackML_Sts.sts_Completing_SC) OR ("PackML".Sts.State.Stopping AND "UN".PackML_Sts.sts_Stopping_SC) OR ("PackML".Sts.State.Aborting AND "UN".PackML_Sts.sts_Aborting_SC) THEN
       #statPackML_CMD_SC := TRUE;
   END_IF;
END_REGION

REGION Network 19: PackML Diagnostics Information to HMI (from LPMLV30 library)
   RUNG wire#powerrail
      Move(in := "HMI_Data".diagnosticsBufferIndexForHMI, out1 => #tempDiagnosticsBufferIndexForHMI)
   END_RUNG
   RUNG wire#powerrail
      { S7_Templates := "SrcType := Int" } LT_Contact(in1 := #tempDiagnosticsBufferIndexForHMI, in2 := 0)
      Move(in := "LPMLV30_DIAG_BUFFER_UPPER_LIM", out1 => #tempDiagnosticsBufferIndexForHMI)
   END_RUNG
   RUNG wire#powerrail
      { S7_Templates := "SrcType := Int" } GT_Contact(in1 := #tempDiagnosticsBufferIndexForHMI, in2 := "LPMLV30_DIAG_BUFFER_UPPER_LIM")
      Move(in := 0, out1 => #tempDiagnosticsBufferIndexForHMI)
   END_RUNG
   RUNG wire#powerrail
      Move(in := "PackML".PackMLDiag.buffer[#tempDiagnosticsBufferIndexForHMI], out1 => "HMI_Data".diagnosticsBufferEntryForHMI)
      Move(in := #tempDiagnosticsBufferIndexForHMI, out1 => "HMI_Data".diagnosticsBufferIndexForHMI)
   END_RUNG
   // the same network as SCL:
   #tempDiagnosticsBufferIndexForHMI := "HMI_Data".diagnosticsBufferIndexForHMI;
   IF #tempDiagnosticsBufferIndexForHMI < 0 THEN
       #tempDiagnosticsBufferIndexForHMI := "LPMLV30_DIAG_BUFFER_UPPER_LIM";
   END_IF;
   IF #tempDiagnosticsBufferIndexForHMI > "LPMLV30_DIAG_BUFFER_UPPER_LIM" THEN
       #tempDiagnosticsBufferIndexForHMI := 0;
   END_IF;
   "HMI_Data".diagnosticsBufferEntryForHMI := "PackML".PackMLDiag.buffer[#tempDiagnosticsBufferIndexForHMI];
   "HMI_Data".diagnosticsBufferIndexForHMI := #tempDiagnosticsBufferIndexForHMI;
END_REGION

REGION Network 20: END: Update the ENO Output. (DO NOT REMOVE. Must be last rung)
   RUNG wire#powerrail
      ReturnCoil( TRUE )
   END_RUNG
   // the same network as SCL:
   ENO := TRUE;
   RETURN;
END_REGION
END_FUNCTION_BLOCK
